{attribute 'hide_all_locals'}
FUNCTION_BLOCK LINAXIS_BECKHOFF EXTENDS FB_3_ROB_AXIS_LIN
VAR_INPUT
	NCAxis : AXIS_REF;
    SETTINGS : stSettings_LinAxis := (
        LinearStandStillLimit := 1.0,
        SafePositionTolerance := 1.0,
        StandardUnits := (
            Position := eUnit.mm,
            Orientation := eUnit.rad,
            Joint := eUnit.mm,
            LinearVelocity := eUnit.mm,
            AngularVelocity := eUnit.rad,
            JointVelocity := eUnit.mm,
            LinearAcceleration := eUnit.mm,
            AngularAcceleration := eUnit.rad,
            JointAcceleration := eUnit.mm));
END_VAR
VAR_IN_OUT
    
END_VAR
VAR_OUTPUT
    AXIS_COMM : FB_3_COMM_AXIS_BECKHOFF;
END_VAR

// ------ CALL CYCLIC -----------------
CYCLIC_LIN_AXIS();
AXIS_COMM(
    Axis := NCAxis,
    StopVelocityTolerance := SETTINGS.LinearStandStillLimit);
COMM := ADR(AXIS_COMM);

// ------ WRITE HMI -------------------
		// NO HMI STRUCT

// ------ READ FROM HMI ---------------
		// NO HMI STRUCT
	


// ------ WRITE PROPS/METHODS ---------
Powered := AXIS_COMM.Powered;
Homed := AXIS_COMM.Homed;
ActualAxisPosition := AXIS_COMM.ActualPosition;
_axisActualVelocity := AXIS_COMM.ActualVelocity;


// ----- CALL POUS AND ERROR SURVEILLANCE ----------


// ----- REST --------------------

METHOD CommandHandler : UINT
VAR_INPUT
    Cmd : eCommands;
    Settings : stCommand_Settings;
END_VAR
VAR
    NewCommandID : UINT;
    TargetPosition : LREAL;
    TargetValid : BOOL;
    EffectiveVelocity : LREAL;
    EffectiveAcceleration : LREAL;
    Accepted : BOOL;
END_VAR
CommandHandler := 0;
IF NOT PrepareAxisCommand(
    Cmd := Cmd,
    Settings := Settings,
    NewCommandID => NewCommandID,
    TargetPosition => TargetPosition,
    TargetValid => TargetValid,
    EffectiveVelocity => EffectiveVelocity,
    EffectiveAcceleration => EffectiveAcceleration) THEN RETURN; END_IF

CASE Cmd OF
    eCommands.MoveL, eCommands.MoveJ, eCommands.MoveJJoints:
        Accepted := AXIS_COMM.SendMoveAbsolute(
            CommandID := NewCommandID,
            Position := TargetPosition,
            Velocity := EffectiveVelocity,
            Acceleration := EffectiveAcceleration,
            Deceleration := SET_A.DefaultDeceleration,
            Jerk := SET_A.DefaultJerk);
    eCommands.MoveLRelativ, eCommands.MoveJRelativ:
        Accepted := AXIS_COMM.SendMoveRelative(
            CommandID := NewCommandID,
            Distance := Settings.Pose.x,
            Velocity := EffectiveVelocity,
            Acceleration := EffectiveAcceleration,
            Deceleration := SET_A.DefaultDeceleration,
            Jerk := SET_A.DefaultJerk);
    eCommands.Homing:
        Accepted := AXIS_COMM.SendHome(CommandID := NewCommandID);
END_CASE

IF Accepted THEN
    CommandHandler := CommitAxisCommand(
        NewCommandID := NewCommandID,
        TargetPosition := TargetPosition,
        TargetValid := TargetValid);
END_IF
END_METHOD

METHOD PROTECTED OnActivate : eResult
VAR
    eParentResult : eResult;
    myResult : eResult;
END_VAR


eParentResult := SUPER^.OnActivate();
myResult := eResult.NONE;

IF eParentResult <> eResult.SUCCESS THEN
    OnActivate := eParentResult;
    RETURN;
END_IF

AXIS_COMM.Power(Enable := FALSE);
IF NOT AXIS_COMM.Powered THEN
    myResult := eResult.SUCCESS;
END_IF

OnActivate := CombineResults(eParentResult, myResult);
END_METHOD

METHOD PROTECTED OnConfigure : eResult
VAR
    eParentResult : eResult;
    myResult : eResult;
END_VAR


eParentResult := SUPER^.OnConfigure();

IF NOT ValidateConfiguration() THEN
    myResult := eResult.FAILURE;
ELSE
    myResult := eResult.SUCCESS;
END_IF

OnConfigure := CombineResults(eParentResult, myResult);
END_METHOD

METHOD PROTECTED OnDeactivate : eResult
VAR
    eParentResult : eResult;
    myResult : eResult;
END_VAR
eParentResult := SUPER^.OnDeactivate();
myResult := eResult.NONE;

IF (ABS(AXIS_COMM.ActualVelocity) > SETTINGS.LinearStandStillLimit) OR AXIS_COMM.Busy THEN
    AXIS_COMM.StopMotion();
ELSE
    AXIS_COMM.Power(Enable := FALSE);
    IF NOT AXIS_COMM.Powered THEN
        myResult := eResult.SUCCESS;
    END_IF
END_IF

OnDeactivate := CombineResults(eParentResult, myResult);
END_METHOD

METHOD PROTECTED OnError : eResult
VAR
    eParentResult : eResult;
    myResult : eResult;
END_VAR
eParentResult := SUPER^.OnError();
myResult := eResult.NONE;


IF eParentResult <> eResult.SUCCESS THEN
    OnError := eParentResult;
    RETURN;
END_IF

IF AXIS_COMM.MESSENGER.HasActivError THEN
    AXIS_COMM.ResetAxis();
    myResult := eResult.NONE;
ELSE
    myResult := eResult.SUCCESS;
END_IF

OnError := CombineResults(eParentResult, myResult);
END_METHOD

END_FUNCTION_BLOCK

(* stored: Version 1.2.0.0, ProductVersion 3.1.4026.18
   POU LINAXIS_BECKHOFF: Id {455244a0-d50f-4d2f-a382-e7e19c641afd}, SpecialFunc None
   Folder StateControl: Id {f6663b81-da1a-49b7-a233-7f100a37ca74}
   Method CommandHandler: Id {d915ac07-9e83-4079-af67-a4609f842e20}
   Method OnActivate: Id {7013f686-7611-45c2-8048-93fa5eb7bab6}
   Method OnConfigure: Id {0c9b9773-f86f-46ad-a92a-7e92d782fa35}
   Method OnDeactivate: Id {5676ee2f-5f23-424a-9aa8-97658c8b66eb}
   Method OnError: Id {a96b6a8d-7acc-40f8-8276-f749a405b545} *)
